TYPE E_CylinderTypeConfig :(
(*Type Configuration of Cylinder*)
	eCylinderType_SINGLE_NORMAL			:=  0,
	eCylinderType_SINGLE_REVERSE 		:=  1,
	eCylinderType_DUEL 					:=  2
);
END_TYPE

(* stored: Version 1.1.0.1, ProductVersion 3.1.4024.2
   DUT E_CylinderTypeConfig: Id {651fcd3c-1456-4089-bbd0-037853552913} *)
